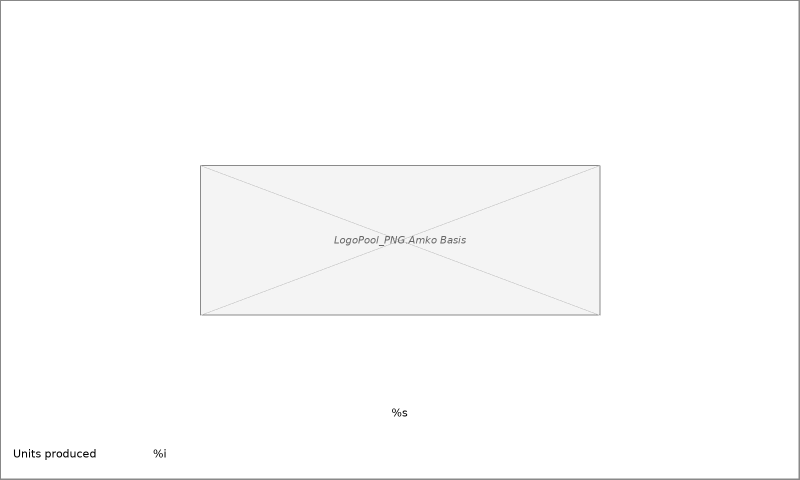
VISUALIZATION LogoScreen_PNG  // 800x480
VAR_INPUT
	nUnitsProduced	: UDINT; // HMI Main total units produced
END_VAR
VAR_IN_OUT
	bCmdManual		: BOOL ; // HMI switch to manual mode
END_VAR
    Frame (0,0 800x480)
        shows ManualButton_PNG(bCmdManual := bCmdManual)
    Image (200,165 400x150), image: LogoPool_PNG.Amko Basis
    Textfield (183,404 433x18), "%s", tooltip "Operator messagages", text variable: GVL_Message.sOPeratorMessage
    Textfield (110,439 100x30), "%i", text variable: nUnitsProduced
    Label (10,439 100x30), "Units produced"
END_VISUALIZATION

(* stored: Version 1.1.0.1, ProductVersion 3.1.4024.5
   Visu LogoScreen_PNG: Id {8e016bc8-ad21-4193-a4ea-5b7cd5d59e25} *)
